(* PLC project Unnamed, Unknown Unnamed 1 *)
(* stored: creationDateTime 2023-06-19T14:42:49, modificationDateTime 2023-06-21T12:42:23 *)

PROGRAM pick_and_place
  VAR
    TP0 : TP;
    CTU0 : CTU;
  END_VAR
  VAR
    ITEM_AT_ENTRY AT %QX0.0 : BOOL;
    ITEM_AT_EXIT AT %QX0.1 : BOOL;
    MOVING_X AT %QX0.2 : BOOL;
    MOVING_Z AT %QX0.3 : BOOL;
    ITEM_DETECTED AT %QX0.4 : BOOL;
    START AT %QX0.5 : BOOL;
    RESET AT %QX0.6 : BOOL;
    STOP AT %QX0.7 : BOOL;
    EMERGENCY_STOP AT %QX1.0 : BOOL;
    AUTO AT %QX1.1 : BOOL;
    FACTORY_IO_RUN AT %QX1.2 : BOOL;
    ENTRY_CONVEYOR AT %QX1.3 : BOOL;
    EXIT_CONVEYOR AT %QX1.4 : BOOL;
    MOVE_X AT %QX1.5 : BOOL;
    MOVE_Z AT %QX1.6 : BOOL;
    GRAB AT %QX1.7 : BOOL;
    START_LIGHT AT %QX2.0 : BOOL;
    RESET_LIGHT AT %QX2.1 : BOOL;
    STOP_LIGHT AT %QX2.2 : BOOL;
    COUNTER AT %QW0 : INT;
  END_VAR
  VAR
    INPUT_STATE : INT := 0;
    I_C_POINT : INT := 0;
    OUTPUT_STATE : INT := 0;
    INPUT_CHANNEL : ARRAY[0..9] OF BOOL;
    OUTPUT_CHANNEL : ARRAY[0..4] OF BOOL;
    T1_DONE : BOOL;
    TIME_DELAY : TIME := t#3s;
    IN_STATE_0 : ARRAY[0..9] OF BOOL := [0, 0, 0, 0, 0, 0, 0, 1, 1, 1];
    IN_STATE_1 : ARRAY[0..9] OF BOOL := [1, 0, 0, 0, 0, 0, 0, 1, 1, 1];
    IN_STATE_2 : ARRAY[0..9] OF BOOL := [1, 0, 0, 0, 0, 1, 1, 1, 1, 1];
    IN_STATE_3 : ARRAY[0..9] OF BOOL := [0, 0, 0, 0, 0, 0, 1, 1, 1, 1];
    IN_STATE_4 : ARRAY[0..9] OF BOOL := [0, 0, 0, 0, 1, 0, 1, 1, 1, 1];
    IN_STATE_5 : ARRAY[0..9] OF BOOL := [0, 1, 0, 0, 1, 1, 1, 1, 1, 1];
    IN_STATE_6 : ARRAY[0..9] OF BOOL := [0, 1, 0, 0, 1, 0, 0, 1, 1, 1];
    OUT_STATE_0 : ARRAY[0..4] OF BOOL := [1, 1, 0, 0, 0];
    OUT_STATE_1 : ARRAY[0..4] OF BOOL := [0, 1, 0, 1, 0];
    OUT_STATE_2 : ARRAY[0..4] OF BOOL := [0, 1, 0, 0, 1];
    OUT_STATE_3 : ARRAY[0..4] OF BOOL := [0, 0, 1, 0, 1];
    OUT_STATE_4 : ARRAY[0..4] OF BOOL := [0, 0, 1, 1, 1];
    OUT_STATE_5 : ARRAY[0..4] OF BOOL := [0, 0, 1, 0, 0];
    OUT_STATE_6 : ARRAY[0..4] OF BOOL := [0, 1, 0, 0, 0];
  END_VAR
  VAR  (* added by the conversion: wires and edge detectors of the diagram *)
    R_TRIG1 : R_TRIG;
  END_VAR

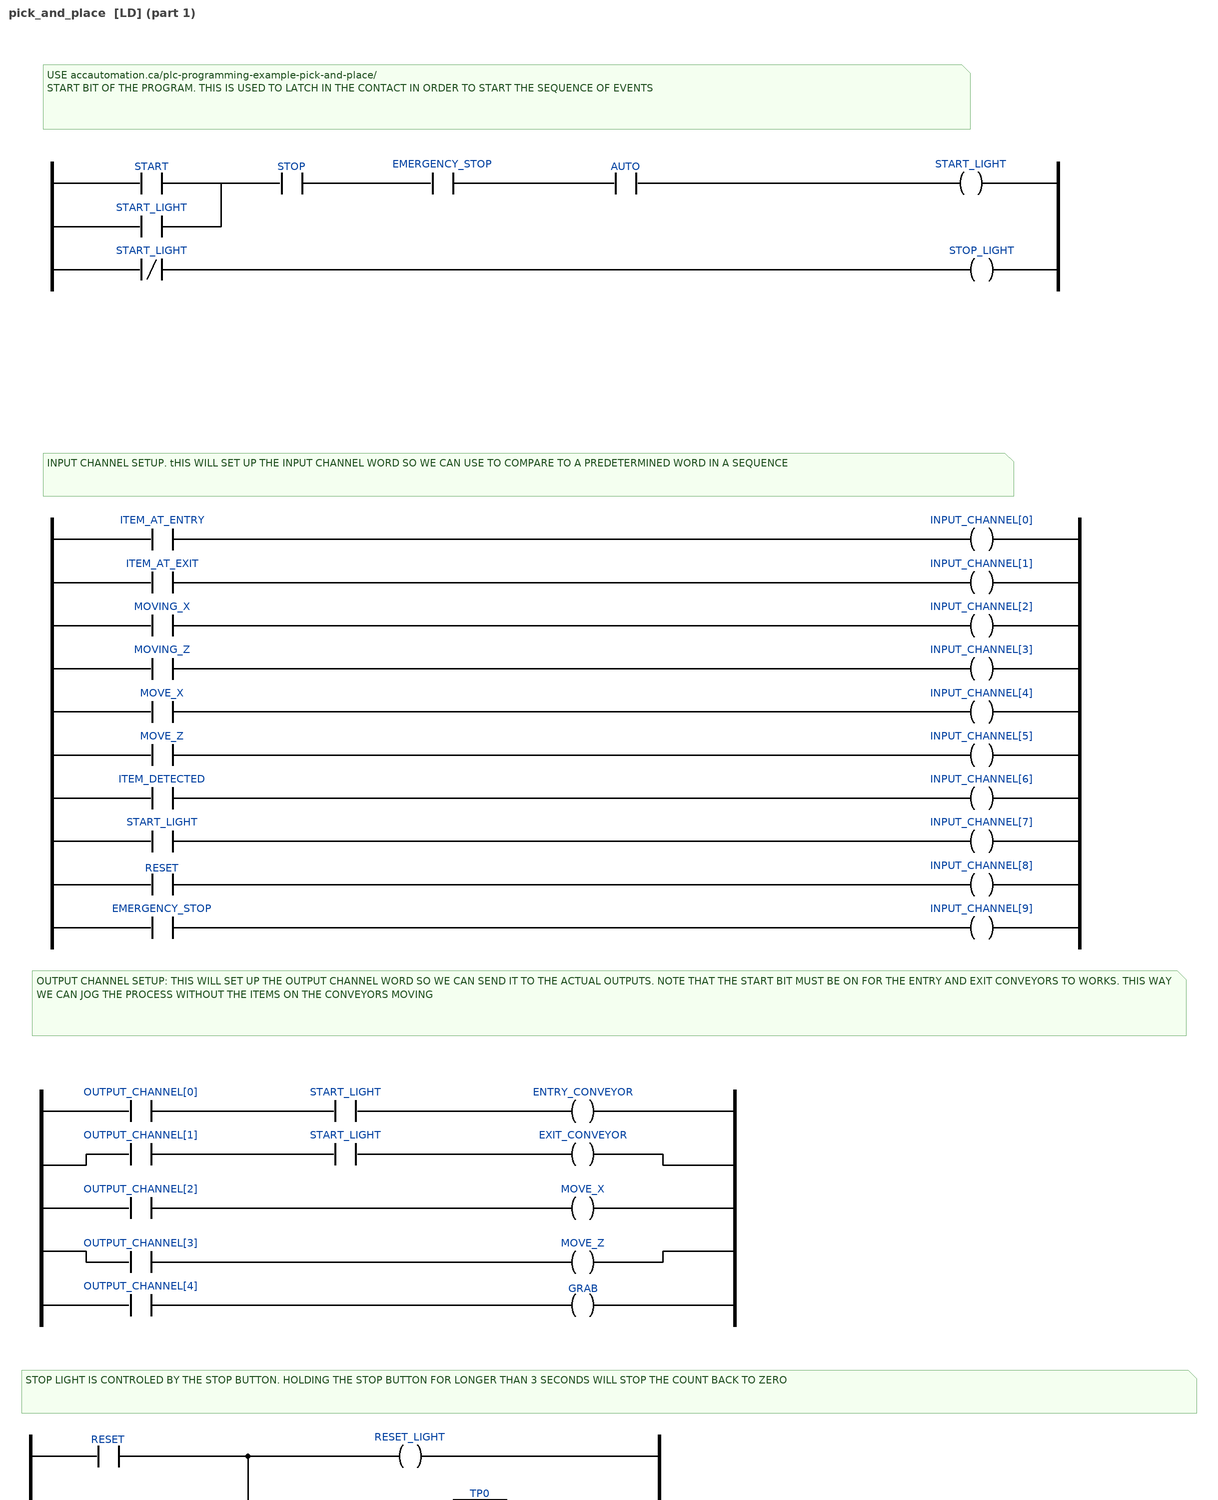
(* LD diagram, written out as Structured Text *)
(* USE accautomation.ca/plc-programming-example-pick-and-place/
START BIT OF THE PROGRAM. THIS IS USED TO LATCH IN THE CONTACT IN ORDER TO START THE SEQUENCE OF EVENTS *)
START_LIGHT := (START OR START_LIGHT) AND STOP AND EMERGENCY_STOP AND AUTO;
STOP_LIGHT := NOT START_LIGHT;
(* INPUT CHANNEL SETUP. tHIS WILL SET UP THE INPUT CHANNEL WORD SO WE CAN USE TO COMPARE TO A PREDETERMINED WORD IN A SEQUENCE *)
INPUT_CHANNEL[0] := ITEM_AT_ENTRY;
INPUT_CHANNEL[1] := ITEM_AT_EXIT;
INPUT_CHANNEL[2] := MOVING_X;
INPUT_CHANNEL[3] := MOVING_Z;
INPUT_CHANNEL[4] := MOVE_X;
INPUT_CHANNEL[5] := MOVE_Z;
INPUT_CHANNEL[6] := ITEM_DETECTED;
INPUT_CHANNEL[7] := START_LIGHT;
INPUT_CHANNEL[8] := RESET;
INPUT_CHANNEL[9] := EMERGENCY_STOP;
(* OUTPUT CHANNEL SETUP: THIS WILL SET UP THE OUTPUT CHANNEL WORD SO WE CAN SEND IT TO THE ACTUAL OUTPUTS. NOTE THAT THE START BIT MUST BE ON FOR THE ENTRY AND EXIT CONVEYORS TO WORKS. THIS WAY WE CAN JOG THE PROCESS WITHOUT THE ITEMS ON THE CONVEYORS MOVING *)
ENTRY_CONVEYOR := OUTPUT_CHANNEL[0] AND START_LIGHT;
EXIT_CONVEYOR := OUTPUT_CHANNEL[1] AND START_LIGHT;
MOVE_X := OUTPUT_CHANNEL[2];
MOVE_Z := OUTPUT_CHANNEL[3];
GRAB := OUTPUT_CHANNEL[4];
(* STOP LIGHT IS CONTROLED BY THE STOP BUTTON. HOLDING THE STOP BUTTON FOR LONGER THAN 3 SECONDS WILL STOP THE COUNT BACK TO ZERO *)
RESET_LIGHT := RESET;
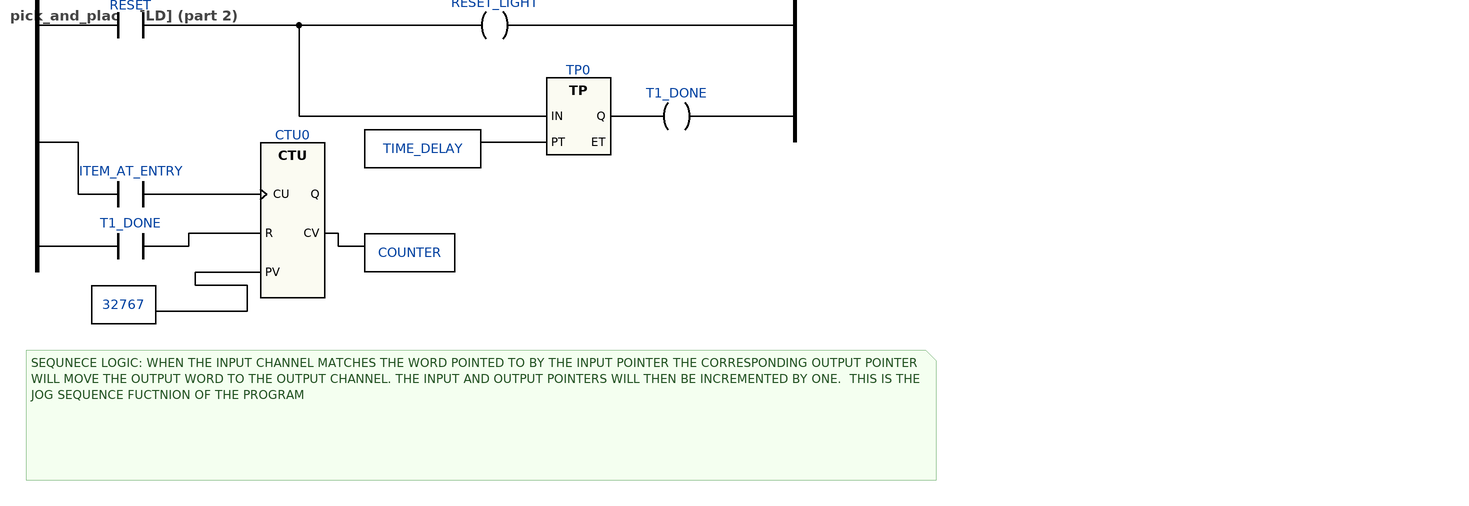
TP0(IN := RESET, PT := TIME_DELAY);
T1_DONE := TP0.Q;
R_TRIG1(CLK := ITEM_AT_ENTRY);
CTU0(CU := R_TRIG1.Q, R := T1_DONE, PV := 32767);
COUNTER := CTU0.CV;
(* SEQUNECE LOGIC: WHEN THE INPUT CHANNEL MATCHES THE WORD POINTED TO BY THE INPUT POINTER THE CORRESPONDING OUTPUT POINTER WILL MOVE THE OUTPUT WORD TO THE OUTPUT CHANNEL. THE INPUT AND OUTPUT POINTERS WILL THEN BE INCREMENTED BY ONE.  THIS IS THE JOG SEQUENCE FUCTNION OF THE PROGRAM *)
END_PROGRAM

FUNCTION_BLOCK FOR_LOOP
  VAR
    INPUT_ARRAY : ARRAY[0..9] OF BOOL;
  END_VAR

            
          
END_FUNCTION_BLOCK

CONFIGURATION Config0
  RESOURCE Res0 ON PLC
    TASK task0(INTERVAL := T#20ms, PRIORITY := 0);
    PROGRAM instance0 WITH task0 : pick_and_place;
  END_RESOURCE
END_CONFIGURATION
